// Mitsubishi GX Works2 project: plcsai   PLC: FX3U/FX3UC

PROGRAM MAIN
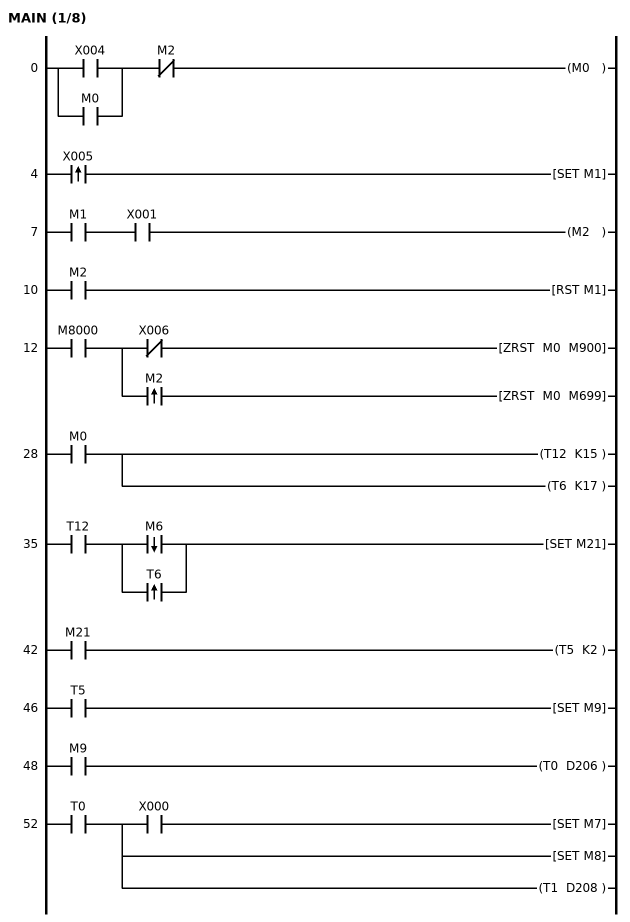
0     LD      X004
      OR      M0
      ANI     M2
      OUT     M0
4     LDP     X005
      SET     M1
7     LD      M1
      AND     X001
      OUT     M2
10    LD      M2
      RST     M1
12    LD      M8000
      MPS
      ANI     X006
      ZRST    M0 M900
      MPP
      ANDP    M2
      ZRST    M0 M699
28    LD      M0
      OUT     T12 K15
      OUT     T6 K17
35    LD      T12
      LDF     M6
      ORP     T6
      ANB
      SET     M21
42    LD      M21
      OUT     T5 K2
46    LD      T5
      SET     M9
48    LD      M9
      OUT     T0 D206
52    LD      T0
      MPS
      AND     X000
      SET     M7
      MPP
      SET     M8
      OUT     T1 D208
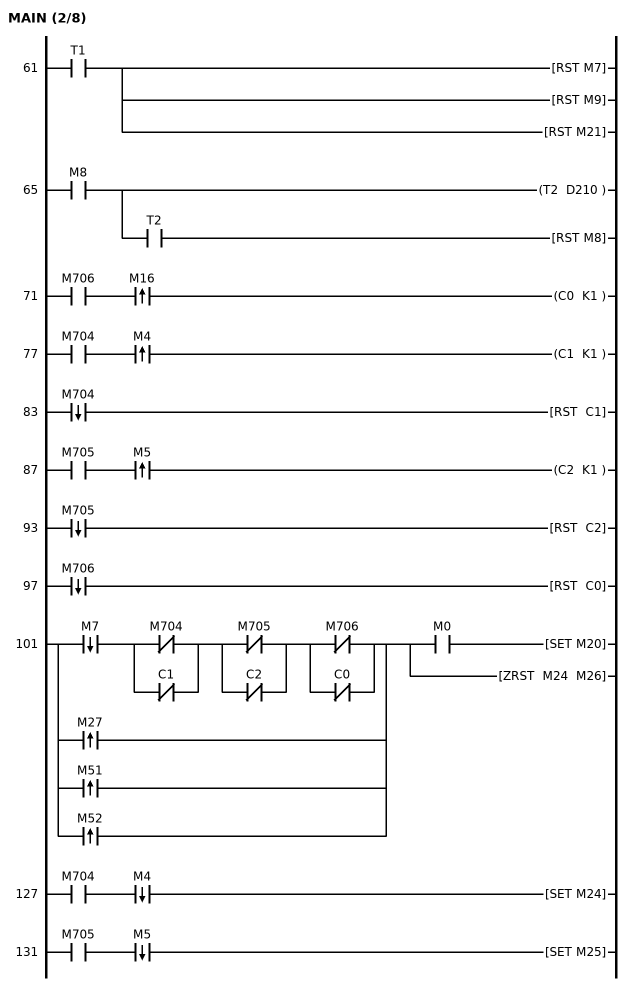
61    LD      T1
      RST     M7
      RST     M9
      RST     M21
65    LD      M8
      OUT     T2 D210
      AND     T2
      RST     M8
71    LD      M706
      ANDP    M16
      OUT     C0 K1
77    LD      M704
      ANDP    M4
      OUT     C1 K1
83    LDF     M704
      RST     C1
87    LD      M705
      ANDP    M5
      OUT     C2 K1
93    LDF     M705
      RST     C2
97    LDF     M706
      RST     C0
101   LDF     M7
      LDI     M704
      ORI     C1
      ANB
      LDI     M705
      ORI     C2
      ANB
      LDI     M706
      ORI     C0
      ANB
      ORP     M27
      ORP     M51
      ORP     M52
      MPS
      AND     M0
      SET     M20
      MPP
      ZRST    M24 M26
127   LD      M704
      ANDF    M4
      SET     M24
131   LD      M705
      ANDF    M5
      SET     M25
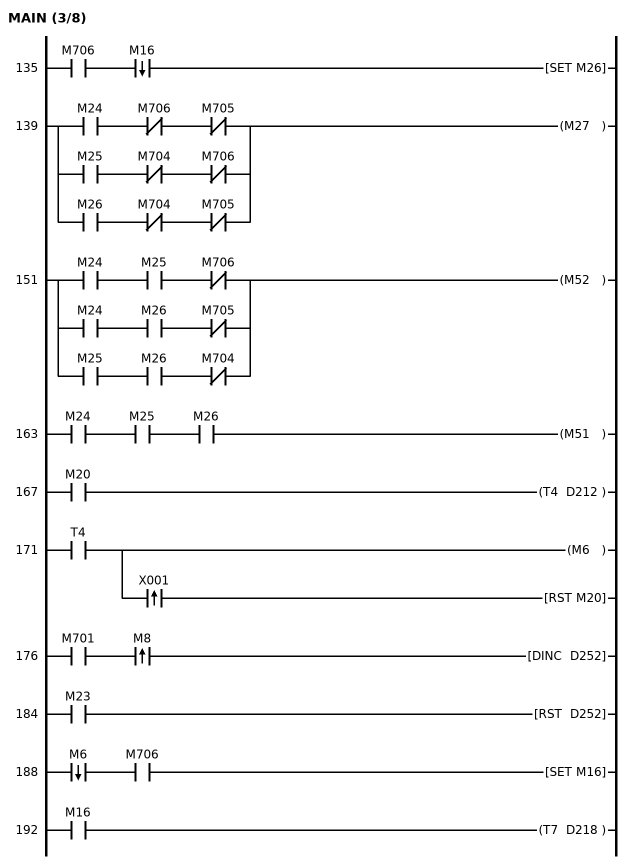
135   LD      M706
      ANDF    M16
      SET     M26
139   LD      M24
      ANI     M706
      ANI     M705
      LD      M25
      ANI     M704
      ANI     M706
      ORB
      LD      M26
      ANI     M704
      ANI     M705
      ORB
      OUT     M27
151   LD      M24
      AND     M25
      ANI     M706
      LD      M24
      AND     M26
      ANI     M705
      ORB
      LD      M25
      AND     M26
      ANI     M704
      ORB
      OUT     M52
163   LD      M24
      AND     M25
      AND     M26
      OUT     M51
167   LD      M20
      OUT     T4 D212
171   LD      T4
      OUT     M6
      ANDP    X001
      RST     M20
176   LD      M701
      ANDP    M8
      DINC    D252
184   LD      M23
      RST     D252
188   LDF     M6
      AND     M706
      SET     M16
192   LD      M16
      OUT     T7 D218
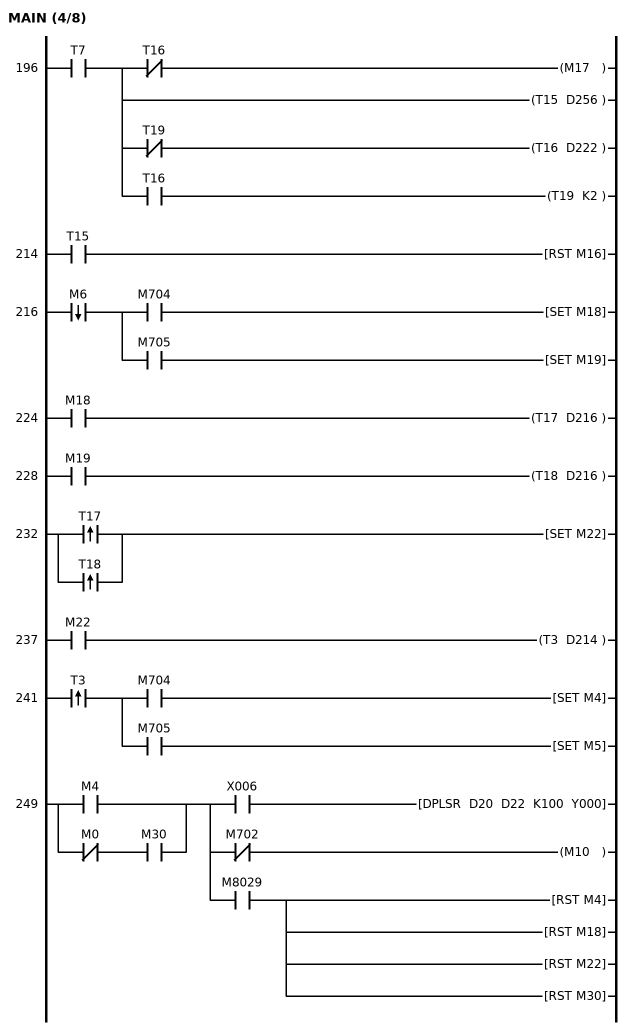
196   LD      T7
      MPS
      ANI     T16
      OUT     M17
      MPP
      OUT     T15 D256
      MPS
      ANI     T19
      OUT     T16 D222
      MPP
      AND     T16
      OUT     T19 K2
214   LD      T15
      RST     M16
216   LDF     M6
      MPS
      AND     M704
      SET     M18
      MPP
      AND     M705
      SET     M19
224   LD      M18
      OUT     T17 D216
228   LD      M19
      OUT     T18 D216
232   LDP     T17
      ORP     T18
      SET     M22
237   LD      M22
      OUT     T3 D214
241   LDP     T3
      MPS
      AND     M704
      SET     M4
      MPP
      AND     M705
      SET     M5
249   LD      M4
      LDI     M0
      AND     M30
      ORB
      MPS
      AND     X006
      DPLSR   D20 D22 K100 Y000
      MRD
      ANI     M702
      OUT     M10
      MPP
      AND     M8029
      RST     M4
      RST     M18
      RST     M22
      RST     M30
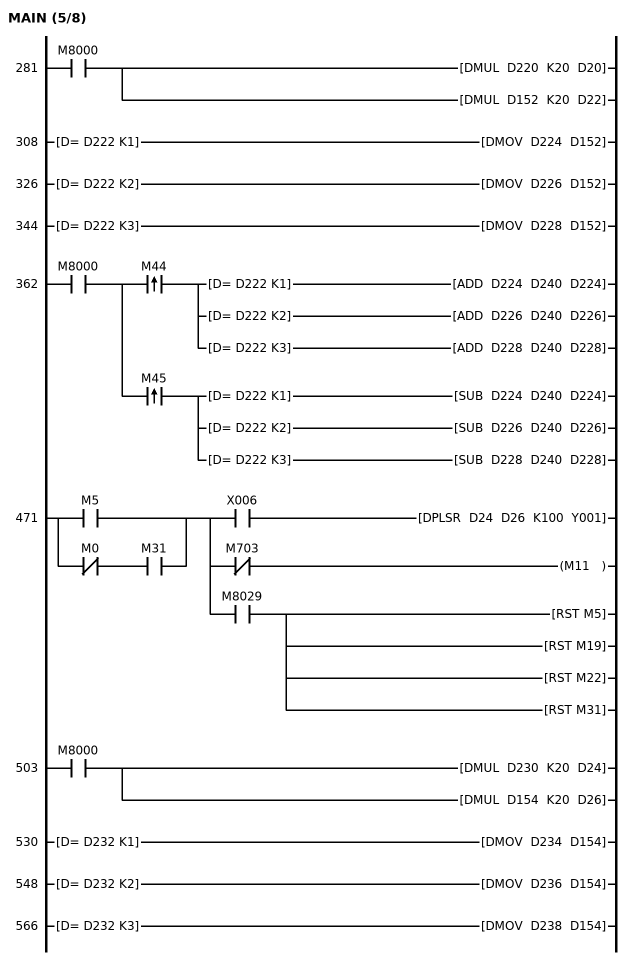
281   LD      M8000
      DMUL    D220 K20 D20
      DMUL    D152 K20 D22
308   LDD=    D222 K1
      DMOV    D224 D152
326   LDD=    D222 K2
      DMOV    D226 D152
344   LDD=    D222 K3
      DMOV    D228 D152
362   LD      M8000
      MPS
      ANDP    M44
      MPS
      ANDD=   D222 K1
      ADD     D224 D240 D224
      MRD
      ANDD=   D222 K2
      ADD     D226 D240 D226
      MPP
      ANDD=   D222 K3
      ADD     D228 D240 D228
      MPP
      ANDP    M45
      MPS
      ANDD=   D222 K1
      SUB     D224 D240 D224
      MRD
      ANDD=   D222 K2
      SUB     D226 D240 D226
      MPP
      ANDD=   D222 K3
      SUB     D228 D240 D228
471   LD      M5
      LDI     M0
      AND     M31
      ORB
      MPS
      AND     X006
      DPLSR   D24 D26 K100 Y001
      MRD
      ANI     M703
      OUT     M11
      MPP
      AND     M8029
      RST     M5
      RST     M19
      RST     M22
      RST     M31
503   LD      M8000
      DMUL    D230 K20 D24
      DMUL    D154 K20 D26
530   LDD=    D232 K1
      DMOV    D234 D154
548   LDD=    D232 K2
      DMOV    D236 D154
566   LDD=    D232 K3
      DMOV    D238 D154
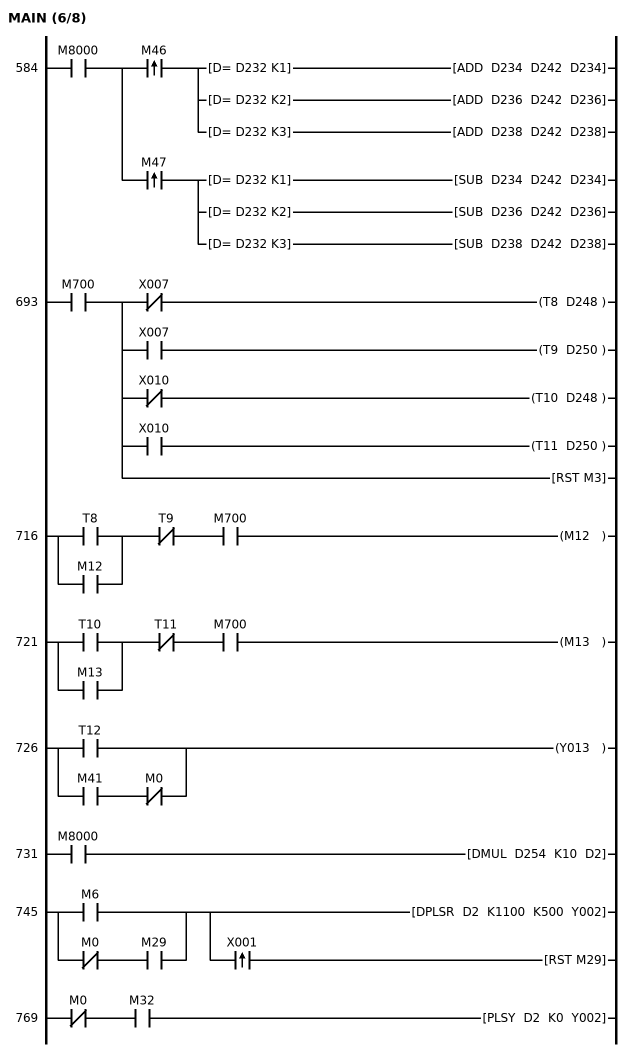
584   LD      M8000
      MPS
      ANDP    M46
      MPS
      ANDD=   D232 K1
      ADD     D234 D242 D234
      MRD
      ANDD=   D232 K2
      ADD     D236 D242 D236
      MPP
      ANDD=   D232 K3
      ADD     D238 D242 D238
      MPP
      ANDP    M47
      MPS
      ANDD=   D232 K1
      SUB     D234 D242 D234
      MRD
      ANDD=   D232 K2
      SUB     D236 D242 D236
      MPP
      ANDD=   D232 K3
      SUB     D238 D242 D238
693   LD      M700
      MPS
      ANI     X007
      OUT     T8 D248
      MRD
      AND     X007
      OUT     T9 D250
      MRD
      ANI     X010
      OUT     T10 D248
      MRD
      AND     X010
      OUT     T11 D250
      MPP
      RST     M3
716   LD      T8
      OR      M12
      ANI     T9
      AND     M700
      OUT     M12
721   LD      T10
      OR      M13
      ANI     T11
      AND     M700
      OUT     M13
726   LD      T12
      LD      M41
      ANI     M0
      ORB
      OUT     Y013
731   LD      M8000
      DMUL    D254 K10 D2
745   LD      M6
      LDI     M0
      AND     M29
      ORB
      DPLSR   D2 K1100 K500 Y002
      ANDP    X001
      RST     M29
769   LDI     M0
      AND     M32
      PLSY    D2 K0 Y002
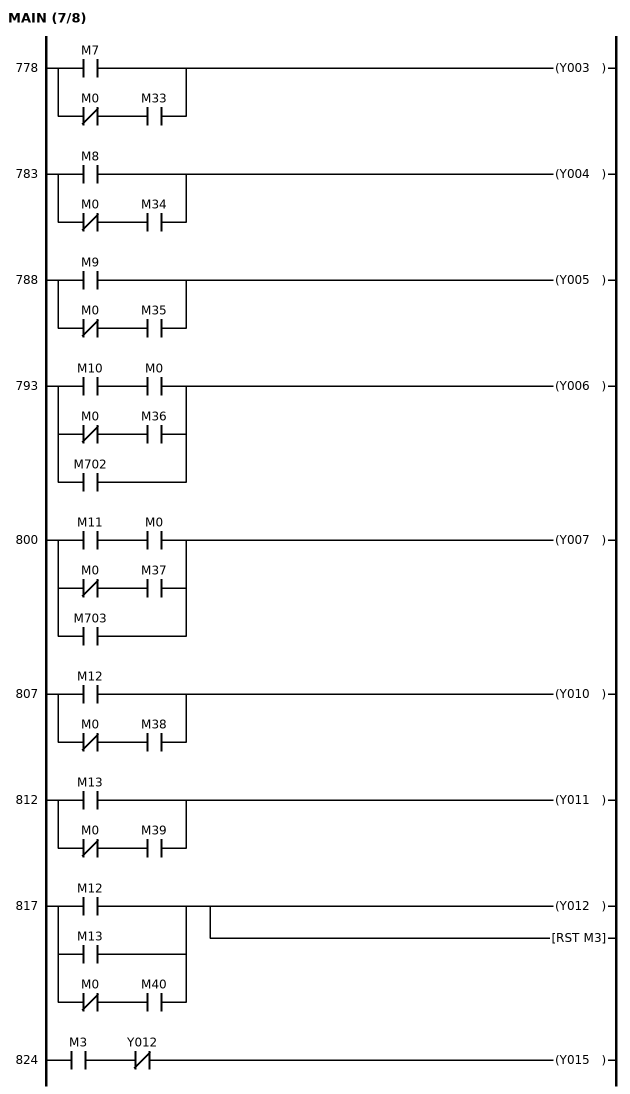
778   LD      M7
      LDI     M0
      AND     M33
      ORB
      OUT     Y003
783   LD      M8
      LDI     M0
      AND     M34
      ORB
      OUT     Y004
788   LD      M9
      LDI     M0
      AND     M35
      ORB
      OUT     Y005
793   LD      M10
      AND     M0
      LDI     M0
      AND     M36
      ORB
      OR      M702
      OUT     Y006
800   LD      M11
      AND     M0
      LDI     M0
      AND     M37
      ORB
      OR      M703
      OUT     Y007
807   LD      M12
      LDI     M0
      AND     M38
      ORB
      OUT     Y010
812   LD      M13
      LDI     M0
      AND     M39
      ORB
      OUT     Y011
817   LD      M12
      OR      M13
      LDI     M0
      AND     M40
      ORB
      OUT     Y012
      RST     M3
824   LD      M3
      ANI     Y012
      OUT     Y015
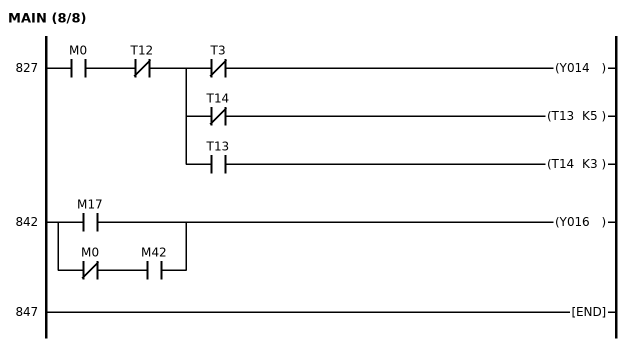
827   LD      M0
      ANI     T12
      MPS
      ANI     T3
      OUT     Y014
      MRD
      ANI     T14
      OUT     T13 K5
      MPP
      AND     T13
      OUT     T14 K3
842   LD      M17
      LDI     M0
      AND     M42
      ORB
      OUT     Y016
847   END
END_PROGRAM
